// TwinCAT 3 PLC project TF6300_FTP_Samples
// Title: TF6300_FTP_Samples
// Company: Beckhoff Automation
// ProjectVersion: 1.0.0
// ProgramVersion: 3.1.4026.11
// libraries:
//   Tc2_FTP, * (Beckhoff Automation GmbH)
//   Tc2_Standard, * (Beckhoff Automation GmbH)
//   Tc2_System, * (Beckhoff Automation GmbH)
//   Tc3_FTP, * (Beckhoff Automation GmbH)
//   Tc3_Module, * (Beckhoff Automation GmbH)
// project tree:
//   DUTs/ E_DoTask.TcDUT
//   / PlcTask.TcTTO
//   POUs/ FB_ManualOperation.TcPOU, FB_SimpleDownload.TcPOU, FB_SimpleUpload.TcPOU, MAIN.TcPOU
// real-time tasks:
//   TASK PlcTask: cycle T#10ms, priority 20, ADS port 350

CONFIGURATION TF6300_FTP_Samples
    RESOURCE PLC ON TwinCAT3
        TASK PlcTask(INTERVAL := T#10ms, PRIORITY := 20);
        PROGRAM MAIN WITH PlcTask : MAIN;
    END_RESOURCE
END_CONFIGURATION

// ---- DUTs/E_DoTask.TcDUT
{attribute 'qualified_only'}
{attribute 'strict'}
TYPE E_DoTask :
(
	NONE := 0,

	CONN_Connect,
	CONN_Disconnect,
	CONN_AddProfile,
	
	EXPLORER_DirExists,
	EXPLORER_DirCreate,
	EXPLORER_DirRemove,
	EXPLORER_DirRename,
	EXPLORER_DirMove,
	
	EXPLORER_FileExists,
	EXPLORER_FileRemove,
	EXPLORER_FileRename,
	EXPLORER_FileMove,
	
	TRANSFER_GetState,
	TRANSFER_GetStateVerbose,
	TRANSFER_Upload,
	TRANSFER_Download,
	TRANSFER_Abort,
	TRANSFER_GetActive,
	TRANSFER_GetActiveVerbose
);
END_TYPE

// ---- POUs/MAIN.TcPOU
PROGRAM MAIN
VAR
	fbSimpleUpload 		: FB_SimpleUpload;
	fbSimpleDownload 	: FB_SimpleDownload;
	fbManualOperation 	: FB_ManualOperation;
END_VAR

fbManualOperation();
fbSimpleUpload();
fbSimpleDownload();

END_PROGRAM

// ---- POUs/FB_SimpleUpload.TcPOU
FUNCTION_BLOCK FB_SimpleUpload
VAR
	bStart 				: BOOL; // Starts the QuickStart sample
	
	fbConnection 		: FB_FtpConnection(1) := (sNetID:= '', tTimeout:= T#60S);
	fbExplorer 			: FB_FtpExplorer := (sNetID:= '', tTimeout:= T#60S);
	fbTransfer 			: FB_FtpTransfer := (sNetID:= '', tTimeout:= T#60S);
	
	stTransferInfo 		: ST_FtpTransferState;
	stNTDataProfile 	: ST_FtpConfigProfile;
	
	sPathToOriginFile 	: STRING(255) := 'C:\Temp\myFileUpload.txt';
	sPathToTargetDir 	: STRING(255) := '\';
	
	bDone 				: BOOL;
	bError 				: BOOL;
	sErrorMSG 			: STRING(255);
	nCase 				: INT;
	nTransferHandle 	: UDINT;
	fbTimer 			: TON := (PT:=T#1S); (* How frequently should the transfer state be checked. Beware of IPC load on very high frequencies. *)
END_VAR

CASE nCase OF
	0: (* Start the QuickStart sample. *)
		IF bStart THEN
			bDone := FALSE;
    		bStart := FALSE;
    		nCase := 10;
		END_IF
		
	10: (* Connect to server by specifying the profile. Create a new profile if the connection profile does not exist, yet. *)
    	IF fbConnection.Connect(
			sFtpConfigProfileFileName:='QuickStart'
		) THEN
			nCase := 15;
    	END_IF
		
	11: (* Connection profile does not exist, yet. Specify connection parameters and store in a new profile. *)
		stNTDataProfile.stConnection.eAuth := E_FtpConnectionAuth.sftp_user_pwd;
		stNTDataProfile.stConnection.nPort := 23;
		stNTDataProfile.stConnection.sHostname := '127.0.0.1';
		stNTDataProfile.stConnection.sUsername := 'My_SFTP_User';
		stNTDataProfile.stConnection.sPassword := 'SomeSecurePassword##1';
		stNTDataProfile.stConnection.sFileName := 'QuickStart';
		
		IF fbConnection.AddProfile(
			stFtpConfigProfile := stNTDataProfile
		) THEN
			nCase := 16;
		END_IF

	15: (* Check connection establishment for any errors. *)
		IF fbConnection.bError THEN
			IF fbConnection.ipResultMessage.EqualsToEventClass(Global.TC_EVENT_CLASSES.TcFtpClientEventClass) THEN
				CASE fbConnection.ipResultMessage.nEventId OF
					E_FtpClientErrorCode.Code_1101_HostConnectionOpen: (* Already connected to the correct host, continue*)
						nCase := 20;
					E_FtpClientErrorCode.Code_1100_AnyConnectionOpen: (* Already connected to another host. Abort.*)
						nCase := 210;
					E_FtpClientErrorCode.Code_1102_FileLocationError: (* Profile has not been created yet. *)
						nCase := 11;
				ELSE
					nCase := 210; (* an unexpected FtpClient error has occured *)
				END_CASE
			ELSE
				nCase := 210; (* an unexpected other error (Ads, Router, ...) has occured*) 
			END_IF
		ELSE
			nCase := 20; (* Start file upload. *)
		END_IF

	16: (* Check profile creation for any errors *)
		IF fbConnection.bError THEN
			IF fbConnection.ipResultMessage.EqualsToEventClass(Global.TC_EVENT_CLASSES.TcFtpClientEventClass) THEN
				CASE fbConnection.ipResultMessage.nEventId OF
					E_FtpClientErrorCode.Code_1106_ParametersImproper: (* The profile is configured improperly (e.g. HostName empty or Port 0) *)
						nCase := 210;
				ELSE
					nCase := 210; (* an unexpected FtpClient error has occured *)
				END_CASE
			ELSE
				nCase := 210; (* an unexpected other error (Ads, Router, ...) has occured*) 
			END_IF
		ELSE
			(* now that the profile has been created, try connecting again *)
			nCase := 10;
		END_IF 

	20: (* Initiate file upload. *)
		IF fbTransfer.Upload(
			fbFtpConnection 		:= fbConnection, 
			sLocalSourcePath 		:= sPathToOriginFile,	
			sServerTargetDirectory 	:= sPathToTargetDir,
			nTransferHandle 		=> nTransferHandle
		) THEN
			nCase := 25;
		END_IF

	25: (* Check file upload initiation for any errors*)
		IF fbTransfer.bError THEN
			IF fbTransfer.ipResultMessage.EqualsToEventClass(Global.TC_EVENT_CLASSES.TcFtpClientEventClass) THEN
				CASE fbTransfer.ipResultMessage.nEventId OF
					E_FtpClientErrorCode.Code_1106_ParametersImproper: (* Source or Target could be empty *)
						nCase := 210;
					E_FtpClientErrorCode.Code_1110_Busy_TryAgain: (* The connection is busy (ONLY FTP). Try again later. *)
						nCase := 210;
				ELSE
					nCase := 210; (* an unexpected FtpClient error has occured *)
				END_CASE
			ELSE
				nCase := 210; (* an unexpected other error (Ads, Router, ...) has occured*) 
			END_IF
		ELSE
			(* now that the transfer has been initialised, check transfer state *)
			nCase := 30;
		END_IF 
		
	30: (* File upload has been started, now cyclically check transfer state. *)
		fbTimer(IN:=TRUE); 
		IF fbTimer.Q THEN
			fbTimer(IN:=FALSE);
			nCase := 40;
		END_IF

	40: (* Request transfer state *)
		IF fbTransfer.GetState(
			fbFtpConnection 		:= fbConnection,
			nTransferHandle 		:= nTransferHandle,
			stTransferState			=> stTransferInfo
		) THEN
			nCase := 45;
		END_IF
		
	45: (* Check GetState for any errors*)
		IF fbTransfer.bError THEN
			IF fbTransfer.ipResultMessage.EqualsToEventClass(Global.TC_EVENT_CLASSES.TcFtpClientEventClass) THEN
				CASE fbTransfer.ipResultMessage.nEventId OF
					E_FtpClientErrorCode.Code_1106_ParametersImproper: (* The transfer for the provided handle could not be found *)
						nCase := 210;
				ELSE
					nCase := 210; (* an unexpected FtpClient error has occured *)
				END_CASE
			ELSE
				nCase := 210; (* an unexpected other error (Ads, Router, ...) has occured*) 
			END_IF
		ELSE
			nCase := 50;
		END_IF

	50: (* Check if file transfer is completed and has not produced any errors *)
		IF (stTransferInfo.eProblem = E_FtpTransferProblemType.None) AND (stTransferInfo.eStep = E_FtpTransferStep.TransferCompleted) THEN
			nCase := 60; // file transfer completed with no errors
		ELSIF stTransferInfo.eProblem <> E_FtpTransferProblemType.None THEN
			nCase := 210; //file transfer encountered an error
		ELSE
			nCase := 30; // not completed yet, check state again
		END_IF
		
	60: (* Disconnect from server. *)
		IF fbConnection.Disconnect() THEN
			nCase := 65;
		END_IF
		
	65: (* Check disconnect for any errors *)
		IF fbConnection.bError THEN
			nCase := 200; (* continue, but warn user that something happened on disconnect *)
		ELSE
			nCase := 70; (* All clear, connection terminated. *)
		END_IF 

	70: (* File upload completed. *)
		bDone := TRUE;
		nCase := 0;

	200: (* File upload completed but unexpected error on disconnect from server. *)
		bDone := TRUE;
		bError := TRUE;
		sErrorMSG := 'Upload was completed successfully, but received error on disconnect. Check [fbConnection.ipResultMessage] for details.';
		nCase := 0;

	210: (* An error has occured. *)
		bDone := TRUE;
		bError := TRUE;
		sErrorMSG := 'Failed to Upload. Check [fbConnection.ipResultMessage] and [stTransferInfo.eProblem]';
		nCase := 0;

END_CASE

END_FUNCTION_BLOCK

// ---- POUs/FB_SimpleDownload.TcPOU
FUNCTION_BLOCK FB_SimpleDownload
VAR
  	bStart 				: BOOL; // Starts the sample
  	
  	fbConnection 		: FB_FtpConnection(1) := (sNetID:= '', tTimeout:= T#60S);
  	fbExplorer 			: FB_FtpExplorer := (sNetID:= '', tTimeout:= T#60S);
  	fbTransfer 			: FB_FtpTransfer := (sNetID:= '', tTimeout:= T#60S);
  	
  	stTransferInfo 		: ST_FtpTransferState;
  	stNTDataProfile 	: ST_FtpConfigProfile;
  	
  	sPathToOriginFile 	: STRING(255) := '\myFileDownload.txt';
  	sPathToTargetDir 	: STRING(255) := 'C:\temp';
  	
  	bDone 				: BOOL;
  	bError 				: BOOL;
  	sErrorMSG 			: STRING(255);
  	nCase 				: INT;
  	nTransferHandle 	: UDINT;
  	fbTimer 			: TON := (PT:=T#1S); (* How frequently should the transfer state be checked. Beware of IPC load on very high frequencies. *)
END_VAR

CASE nCase OF
	0: (* Start the sample. *)
		IF bStart THEN
			bDone := FALSE;
    		bStart := FALSE;
    		nCase := 10;
		END_IF
		
	10: (* Connect to server by specifying the profile. Create a new profile if the connection profile does not exist, yet. *)
    	IF fbConnection.Connect(
			sFtpConfigProfileFileName:='QuickStart'
		) THEN
			nCase := 15;
    	END_IF
		
	11: (* Connection profile does not exist, yet. Specify connection parameters and store in a new profile. *)
		stNTDataProfile.stConnection.eAuth := E_FtpConnectionAuth.sftp_user_pwd;
		stNTDataProfile.stConnection.nPort := 23;
		stNTDataProfile.stConnection.sHostname := '127.0.0.1';
		stNTDataProfile.stConnection.sUsername := 'My_SFTP_User';
		stNTDataProfile.stConnection.sPassword := 'SomeSecurePassword##1';
		stNTDataProfile.stConnection.sFileName := 'QuickStart';
		
		IF fbConnection.AddProfile(
			stFtpConfigProfile := stNTDataProfile
		) THEN
			nCase := 16;
		END_IF

	15: (* Check connection establishment for any errors. *)
		IF fbConnection.bError THEN
			IF fbConnection.ipResultMessage.EqualsToEventClass(Global.TC_EVENT_CLASSES.TcFtpClientEventClass) THEN
				CASE fbConnection.ipResultMessage.nEventId OF
					E_FtpClientErrorCode.Code_1101_HostConnectionOpen: (* Already connected to the correct host, continue*)
						nCase := 20;
					E_FtpClientErrorCode.Code_1100_AnyConnectionOpen: (* Already connected to another host. Abort.*)
						nCase := 210;
					E_FtpClientErrorCode.Code_1102_FileLocationError: (* Profile has not been created yet. *)
						nCase := 11;
				ELSE
					nCase := 210; (* an unexpected FtpClient error has occured *)
				END_CASE
			ELSE
				nCase := 210; (* an unexpected other error (Ads, Router, ...) has occured*) 
			END_IF
		ELSE
			nCase := 20; (* Start file upload. *)
		END_IF

	16: (* Check profile creation for any errors *)
		IF fbConnection.bError THEN
			IF fbConnection.ipResultMessage.EqualsToEventClass(Global.TC_EVENT_CLASSES.TcFtpClientEventClass) THEN
				CASE fbConnection.ipResultMessage.nEventId OF
					E_FtpClientErrorCode.Code_1106_ParametersImproper: (* The profile is configured improperly (e.g. HostName empty or Port 0) *)
						nCase := 210;
				ELSE
					nCase := 210; (* an unexpected FtpClient error has occured *)
				END_CASE
			ELSE
				nCase := 210; (* an unexpected other error (Ads, Router, ...) has occured*) 
			END_IF
		ELSE
			(* now that the profile has been created, try connecting again *)
			nCase := 10;
		END_IF 

	20: (* Initiate file upload. *)
		IF fbTransfer.Download(
			fbFtpConnection 		:= fbConnection, 
			sServerSourcePath 		:= sPathToOriginFile,	
			sLocalTargetDirectory  	:= sPathToTargetDir,
			nTransferHandle 		=> nTransferHandle
		) THEN
			nCase := 25;
		END_IF

	25: (* Check file upload initiation for any errors*)
		IF fbTransfer.bError THEN
			IF fbTransfer.ipResultMessage.EqualsToEventClass(Global.TC_EVENT_CLASSES.TcFtpClientEventClass) THEN
				CASE fbTransfer.ipResultMessage.nEventId OF
					E_FtpClientErrorCode.Code_1106_ParametersImproper: (* Source or Target could be empty *)
						nCase := 210;
					E_FtpClientErrorCode.Code_1110_Busy_TryAgain: (* The connection is busy (ONLY FTP). Try again later. *)
						nCase := 210;
				ELSE
					nCase := 210; (* an unexpected FtpClient error has occured *)
				END_CASE
			ELSE
				nCase := 210; (* an unexpected other error (Ads, Router, ...) has occured*) 
			END_IF
		ELSE
			(* now that the transfer has been initialised, check transfer state *)
			nCase := 30;
		END_IF 
		
	30: (* File upload has been started, now cyclically check transfer state. *)
		fbTimer(IN:=TRUE); 
		IF fbTimer.Q THEN
			fbTimer(IN:=FALSE);
			nCase := 40;
		END_IF

	40: (* Request transfer state *)
		IF fbTransfer.GetState(
			fbFtpConnection 		:= fbConnection,
			nTransferHandle 		:= nTransferHandle,
			stTransferState			=> stTransferInfo
		) THEN
			nCase := 45;
		END_IF
		
	45: (* Check GetState for any errors*)
		IF fbTransfer.bError THEN
			IF fbTransfer.ipResultMessage.EqualsToEventClass(Global.TC_EVENT_CLASSES.TcFtpClientEventClass) THEN
				CASE fbTransfer.ipResultMessage.nEventId OF
					E_FtpClientErrorCode.Code_1106_ParametersImproper: (* The transfer for the provided handle could not be found *)
						nCase := 210;
				ELSE
					nCase := 210; (* an unexpected FtpClient error has occured *)
				END_CASE
			ELSE
				nCase := 210; (* an unexpected other error (Ads, Router, ...) has occured*) 
			END_IF
		ELSE
			nCase := 50;
		END_IF

	50: (* Check if file transfer is completed and has not produced any errors *)
		IF (stTransferInfo.eProblem = E_FtpTransferProblemType.None) AND (stTransferInfo.eStep = E_FtpTransferStep.TransferCompleted) THEN
			nCase := 60; // file transfer completed with no errors
		ELSIF stTransferInfo.eProblem <> E_FtpTransferProblemType.None THEN
			nCase := 210; //file transfer encountered an error
		ELSE
			nCase := 30; // not completed yet, check state again
		END_IF
		
	60: (* Disconnect from server. *)
		IF fbConnection.Disconnect() THEN
			nCase := 65;
		END_IF
		
	65: (* Check disconnect for any errors *)
		IF fbConnection.bError THEN
			nCase := 200; (* continue, but warn user that something happened on disconnect *)
		ELSE
			nCase := 70; (* All clear, connection terminated. *)
		END_IF 

	70: (* File upload completed. *)
		bDone := TRUE;
		nCase := 0;

	200: (* File upload completed but unexpected error on disconnect from server. *)
		bDone := TRUE;
		bError := TRUE;
		sErrorMSG := 'Download was completed successfully, but received error on disconnect. Check [fbConnection.ipResultMessage] for details.';
		nCase := 0;

	210: (* An error has occured. *)
		bDone := TRUE;
		bError := TRUE;
		sErrorMSG := 'Failed to Download. Check [fbConnection.ipResultMessage] and [stTransferInfo.eProblem]';
		nCase := 0;

END_CASE

END_FUNCTION_BLOCK

// ---- POUs/FB_ManualOperation.TcPOU
FUNCTION_BLOCK FB_ManualOperation
VAR
	fbConnection 	: FB_FtpConnection(1) 	:= (sNetID := '', tTimeout := T#50S);
	fbExplorer		: FB_FtpExplorer 		:= (sNetID := '', tTimeout := T#50S);
	fbTransfer 		: FB_FtpTransfer 		:= (sNetID := '', tTimeout := T#50S);

	stConfigProfile: ST_FtpConfigProfile := (
		stConnection := (
			eAuth := E_FtpConnectionAuth.sftp_user_pwd, 
			nPort := 23, 
			sHostname := '127.0.0.1', 
			sUsername := 'My_SFTP_User', 
			sPassword := 'SomeSecurePassword##1', 
			sFileName := 'QuickStart')
	);
	
    sLocalDirectory			: STRING(255) := 'C:\temp\';
	sRemoteDirectory		: STRING(255) := '\';
	sNewRemoteDirectory		: STRING(255) := '\';
	sLocalFilePath			: STRING(255) := 'C:\temp\file.txt';
	sRemoteFilePath			: STRING(255) := '\file.txt';
	sNewName				: STRING(255) := 'NewElementName';
	
	stTransferState			: ST_FtpTransferState;
	stTransferStateVerbose	: ST_FtpTransferStateVerbose;
	
	stTransfersActive		: ST_FtpTransfersActive;
	aTransfersActiveList	: A_FtpTransfersActiveList;
	
	bFileExists				: BOOL;
	bDirExists				: BOOL;
		
	nHandle					: UDINT;
	eDoTask					: E_DoTask := E_DoTask.NONE;
END_VAR

CASE eDoTask OF
// ====================================================================================================================================	
//	Actions that make use of FB_FTP_Connection alias fbCONNECTION
// ==================================================================================================================================== 		
		
	E_DoTask.CONN_Connect:
		IF fbConnection.Connect(stConfigProfile.stConnection.sFileName) THEN
			eDoTask := E_DoTask.NONE;	
		END_IF
	
	E_DoTask.CONN_Disconnect:
		IF fbConnection.Disconnect() THEN
			eDoTask := E_DoTask.NONE;
		END_IF
		
	E_DoTask.CONN_AddProfile:
		IF fbConnection.AddProfile(stConfigProfile) THEN
			eDoTask := E_DoTask.NONE;
		END_IF
	
// ====================================================================================================================================	
//	Actions that make use of FB_FTP_Explorer alias fbEXPLORER
// ==================================================================================================================================== 

// ============================================================ Directories =========================================================== 
		
	E_DoTask.EXPLORER_DirCreate:
		IF fbExplorer.DirCreate(fbConnection, sRemoteDirectory) THEN
			eDoTask := E_DoTask.NONE;
		END_IF
	
	E_DoTask.EXPLORER_DirExists:
		IF fbExplorer.DirExists(fbConnection, sRemoteDirectory, bExists => bDirExists) THEN		
	    	eDoTask := E_DoTask.NONE;	
		END_IF
	
	E_DoTask.EXPLORER_DirRemove:
		IF fbExplorer.DirRemove(fbConnection, sRemoteDirectory) THEN
			eDoTask := E_DoTask.NONE;
		END_IF
	
	E_DoTask.EXPLORER_DirRename:
		IF fbExplorer.DirRename(fbConnection, sRemoteDirectory, sNewName) THEN
			eDoTask := E_DoTask.NONE;
		END_IF
		
	E_DoTask.EXPLORER_DirMove:
		IF fbExplorer.DirMove(fbConnection, sRemoteDirectory, sNewRemoteDirectory) THEN
			eDoTask := E_DoTask.NONE;
		END_IF
		
// =============================================================== Files ============================================================== 
		
	E_DoTask.EXPLORER_FileExists:
		IF fbExplorer.FileExists(fbConnection, sRemoteFilePath, bExists => bFileExists) THEN
			eDoTask := E_DoTask.NONE;
		END_IF
		
	E_DoTask.EXPLORER_FileRemove:
		IF fbExplorer.FileRemove(fbConnection, sRemoteFilePath) THEN
			eDoTask := E_DoTask.NONE;
		END_IF
	
	E_DoTask.EXPLORER_FileRename:
		IF fbExplorer.FileRename(fbConnection, sRemoteFilePath, sNewName) THEN
			eDoTask := E_DoTask.NONE;
		END_IF
		
	E_DoTask.EXPLORER_FileMove:
		IF fbExplorer.FileMove(fbConnection, sRemoteFilePath, sNewRemoteDirectory) THEN
			eDoTask := E_DoTask.NONE;
		END_IF
		
// ====================================================================================================================================	
//	Actions that make use of FB_FTP_Transfer alias fbTRANSFER
// ==================================================================================================================================== 
		
	E_DoTask.TRANSFER_Download:
		IF fbTransfer.Download(fbConnection, sRemoteFilePath, sLocalDirectory, nTransferHandle => nHandle) THEN
			eDoTask := E_DoTask.NONE;
		END_IF
		
	E_DoTask.TRANSFER_Upload:
		IF fbTransfer.Upload(fbConnection, sLocalFilePath, sRemoteDirectory, nTransferHandle => nHandle) THEN
			eDoTask := E_DoTask.NONE;
		END_IF
		
	E_DoTask.TRANSFER_GetState:
		IF fbTransfer.GetState(fbConnection, nHandle, stTransferState => stTransferState) THEN
			eDoTask := E_DoTask.NONE;
		END_IF
		
	E_DoTask.TRANSFER_GetStateVerbose:
		IF fbTransfer.GetStateVerbose(fbConnection, nHandle, stTransferStateVerbose => stTransferStateVerbose) THEN
			eDoTask := E_DoTask.NONE;
		END_IF
	
	E_DoTask.TRANSFER_Abort:
		IF fbTransfer.Abort(fbConnection, nHandle) THEN
			eDoTask := E_DoTask.NONE;
		END_IF
		
	E_DoTask.TRANSFER_GetActive:
		IF fbTransfer.GetActive(fbConnection, stTransfers => stTransfersActive) THEN
			eDoTask := E_DoTask.NONE;
		END_IF
		
	E_DoTask.TRANSFER_GetActiveVerbose:
		IF fbTransfer.GetActiveVerbose(fbConnection, stTransfers => stTransfersActive, aTransfersList => aTransfersActiveList) THEN
			eDoTask := E_DoTask.NONE;
		END_IF
END_CASE

END_FUNCTION_BLOCK
